FUNCTION_BLOCK UA_GetNameSpaceIndexWrapper IMPLEMENTS I_OPCUA_GetNameSpaceIndex
VAR_INPUT
END_VAR
VAR_OUTPUT
END_VAR
VAR
	uaGetNameSpaceIndex : UA_GetNameSpaceIndex;
END_VAR

{warning 'add method implementation '}
METHOD start : BOOL
VAR_INPUT
	Execute			: BOOL;
	ConnectionHdl	: DWORD;
	NamespaceUri	: STRING(MAX_STRING_LENGTH);
	Timeout			: TIME := DEFAULT_ADS_TIMEOUT;
END_VAR
VAR_OUTPUT
	NamespaceIndex	: UINT;
	Done			: BOOL;
	Busy			: BOOL;
	Error			: BOOL;
	ErrorID			: DWORD;
END_VAR
uaGetNameSpaceIndex(Execute			:= ,
                    ConnectionHdl	:= ,
                    NamespaceUri	:= ,
                    Timeout			:= ,
					NamespaceIndex	=> ,
                    Done			=> ,
                    Busy			=> ,
                    Error			=> ,
                    ErrorID			=> );
END_METHOD

END_FUNCTION_BLOCK

(* stored: Version 1.1.0.1, ProductVersion 3.1.4024.9
   POU UA_GetNameSpaceIndexWrapper: Id {bfe2eaec-80ee-46fd-93e6-c3ee92cb67ca}, SpecialFunc None
   Method start: Id {6482bda8-fa83-4352-8923-ebd6ac8df001} *)
